(*

.. <legal notes>

legal notes
=================
| SPDX-FileCopyrightText: © 2026 Oleksandr Tiutyk <trofimich@gmail.com>
| SPDX-License-Identifier: LGPL-3.0-only
| For details check: LGPL-3.0-only_

.. _LGPL-3.0-only: https://www.gnu.org/licenses/lgpl-3.0.en.html

.. </legal notes>

*)

INTERFACE ISimpleDevice EXTENDS IDevice

{attribute 'monitoring' := 'call'}
PROPERTY BoundToIO : BOOL
GET
END_GET
END_PROPERTY

END_INTERFACE

(* stored: Version 1.1.0.1
   Itf ISimpleDevice: Id {15135d0b-b078-4046-91ab-232b065f7af4}
   Property BoundToIO: Id {691c29d0-ca9a-4c5e-bbe0-cf1616f7164d}
   Get Get: Id {3e4c77b4-020e-4dd6-a8f9-7b92bef1192c} *)
